FUNCTION_BLOCK CARSIM
VAR_INPUT
	valvePosition : REAL := 0;
	//init : BOOL := FALSE;
	carWt: REAL := 1000;

	scanTime: REAL := 0.05; //milliseconds
	carRollResist : REAL := 0.001; // lbs per ton
	initialize : BOOL;
END_VAR
VAR_IN_OUT
	
	
END_VAR
VAR_OUTPUT
	car : CarPasser;
	incOut : BOOL := FALSE;
END_VAR
VAR
	
END_VAR




IF initialize THEN
	car.vel := 0;
	car.acc := 0;
	car.pos := 0;
	car.accelLoad := 0;
	
	car.velPrev := 0;
	car.accPrev := 0;	
	car.posPrev :=0;
	car.accelLoadPrev:= 0;
	car.carWeight := carWt;
	car.valveFlowEst := 0;
	initialize:=FALSE;
END_IF


car.velPrev := car.vel;
car.accPrev := car.acc;	
car.posPrev := car.pos;
car.accelLoadPrev := car.accelLoad;

IF ABS(valvePosition) > 0.1 THEN
	car.valveFlowEst := 0.0319*EXPT(ABS(valvePosition), 2.0) - 0.1504*ABS(valvePosition) +5.04; // liters/minute
ELSE
	car.valveFlowEst := 0;	
END_IF

//flow negate flow for opposite movement
IF valvePosition < 0 THEN
	car.valveFlowEst := -car.valveFlowEst;
END_IF

car.vel :=  0.0084*car.valveFlowEst;

//OK Just make it not spike
IF ABS(car.vel - car.velPrev)/0.050 > 1.5 THEN
	
	car.acc := 0;
ELSE
	car.acc :=ABS(car.vel - car.velPrev)/0.050;
END_IF
car.pos := car.posPrev + car.vel*0.05; 
car.accelLoad := carRollResist*car.carWeight/2000 + car.carWeight/32.2*car.acc;
car.power := car.accelLoad*60/33000;

END_FUNCTION_BLOCK

(* stored: Version 1.1.0.1
   POU CARSIM: Id {6351b867-5755-4318-9827-0ba11a6c53ee}, SpecialFunc None *)
